FUNCTION_BLOCK ExportRealDataToFile
VAR_INPUT
	arrREALData				: ARRAY[0..Parameters.iArrayREALSize] OF REAL;
	sFilePath				: STRING(255); // File Path
	bUseTimeStamp 			: BOOL;
	bRoundREALDataValues	: BOOL;
	iRoundingDecIndex		: INT := 2; 
	
	bExport					: BOOL;
END_VAR
VAR_OUTPUT
	bExportDone					: BOOL; // Trigger signal for ExportDone
END_VAR
VAR	
	sInputFilePath			: STRING(255);
	// TimeStamp
	timeStamp				: STRING(255);
	sFilePathPlusTimestamp	: STRING(255);
	fbSysTime   			: FB_LocalSystemTime := ( bEnable := TRUE, dwCycle := 1 );
	
	// Export Data
	fbExport 				: ExportArrayREALDataToTextFile;
	
	i						: INT;
END_VAR

// get system time
fbSysTime();

// use time stamp to file name
IF bUseTimeStamp THEN
	// get time stamp
	timeStamp := F_GET_TIME_STAMP(fbSysTime.systemTime, '_', '_');
	sFilePathPlusTimestamp := INSERT(sFilePath,CONCAT('_',timeStamp),FIND(sFilePath, '.txt') - 1);
	sInputFilePath := sFilePathPlusTimestamp;
ELSE
	sInputFilePath := sFilePath;
END_IF

// round array data values
IF bRoundREALDataValues THEN
	FOR i := 0 TO Parameters.iArrayREALSize DO
		arrREALData[i] := F_ROUND_REAL(arrREALData[i], iRoundingDecIndex);
	END_FOR
END_IF


fbExport(
	arrData:= arrREALData, 
	bExecute:= bExport, 
	bUseTimeStamp:= bUseTimeStamp, 
	sFilePath:= sInputFilePath, 
	bDone=> bExportDone);

END_FUNCTION_BLOCK

(* stored: Version 1.1.0.1, ProductVersion 3.1.4024.9
   POU ExportRealDataToFile: Id {018281cf-19ee-4322-9da9-c7dda6984da7}, SpecialFunc None *)
